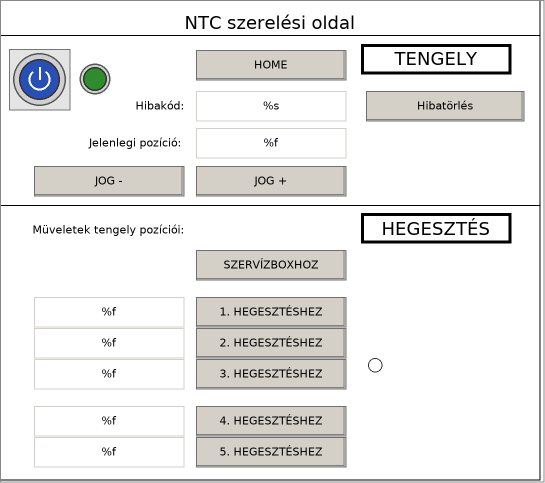
VISUALIZATION Hegesztes_Tengely_NTC  // 545x483
    Rectangle (0,0 540x480)
    PowerSwitch (9,49 61x61), variable: GVL.bJozsiServo, behaviour: TOGGLE, style: Switch-PowerSwitch-Blue
    Button (196,50 150x30), "HOME"
        OnMouseUp: execute { JOZSITENGELY.sJozsiAxisCommand:='HOME'; }
    Button (196,166 150x30), "JOG +"
        tap JOZSITENGELY.bJozsiJOGPlus
    Button (34,166 150x30), "JOG -"
        tap JOZSITENGELY.bJozsiJOGMinus
    Button (366,91 158x30), "Hibatörlés"
        tap JOZSITENGELY.bJozsiReset
    Textfield (196,91 150x30), "%s", text variable: JOZSITENGELY.nJozsiErrorCode, input disabled if: TRUE
    Label (34,128 150x30), "Jelenlegi pozíció:"
    Textfield (196,128 150x30), "%f", text variable: JOZSITENGELY.lrJozsiActPos, input disabled if: TRUE
    Textfield (34,297 150x30), "%f", text variable: GVL.lrHegesztoPosition1
        OnMouseClick: write the text variable via VisuDialogs.Numpad, min -10000, max -1
    Button (196,297 150x30), "1. HEGESZTÉSHEZ"
        OnMouseUp: execute { JOZSITENGELY.lrJozsiPosition:=GVL.lrHegesztoPosition1; JOZSITENGELY.sJozsiAxisCommand:='MOVE'; }
    RadioButton (366,249 177x232), variable: HEGESZTOK.nHegesztoNum
        Areas[0]: Text=Semelyik
        Areas[1]: Text=Program1HG1
        Areas[2]: Text=Program2HG1
        Areas[3]: Text=Program3HG1
        Areas[4]: Text=Program4HG2
        Areas[5]: Text=Program5HG2
        p340057476: Készenléti program
        p3123465237: 1. hegesztés program
        p2481256679: 2. hegesztés program
        p1032612214: 3. hegesztés program
        p3228930307: 4. hegesztés program
        p1847394450: 5. hegesztés program
        p1205187680: Program7HG3
        p3921487345: Program8HG3
    Textfield (34,328 150x30), "%f", text variable: GVL.lrHegesztoPosition2
        OnMouseClick: write the text variable via VisuDialogs.Numpad, min -10000, max -1
    Button (196,328 150x30), "2. HEGESZTÉSHEZ"
        OnMouseUp: execute { JOZSITENGELY.lrJozsiPosition:=GVL.lrHegesztoPosition2; JOZSITENGELY.sJozsiAxisCommand:='MOVE'; }
    Textfield (34,359 150x30), "%f", text variable: GVL.lrHegesztoPosition3
        OnMouseClick: write the text variable via VisuDialogs.Numpad, min -10000, max -1
    Button (196,359 150x30), "3. HEGESZTÉSHEZ"
        OnMouseUp: execute { JOZSITENGELY.lrJozsiPosition:=GVL.lrHegesztoPosition3; JOZSITENGELY.sJozsiAxisCommand:='MOVE'; }
    Textfield (34,406 150x30), "%f", text variable: GVL.lrHegesztoPosition4
        OnMouseClick: write the text variable via VisuDialogs.Numpad, min -10000, max -1
    Button (196,406 150x30), "4. HEGESZTÉSHEZ"
        OnMouseUp: execute { JOZSITENGELY.lrJozsiPosition:=GVL.lrHegesztoPosition4; JOZSITENGELY.sJozsiAxisCommand:='MOVE'; }
    Textfield (34,437 150x30), "%f", text variable: GVL.lrHegesztoPosition5
        OnMouseClick: write the text variable via VisuDialogs.Numpad, min -10000, max -1
    Button (196,437 150x30), "5. HEGESZTÉSHEZ"
        OnMouseUp: execute { JOZSITENGELY.lrJozsiPosition:=GVL.lrHegesztoPosition5; JOZSITENGELY.sJozsiAxisCommand:='MOVE'; }
    Button (196,250 150x30), "SZERVÍZBOXHOZ"
        OnMouseUp: execute { JOZSITENGELY.lrJozsiPosition:=GVL.lrNTCSzervizbox; JOZSITENGELY.sJozsiAxisCommand:='MOVE'; }
    Lamp1 (77,61 36x36), variable: JOZSITENGELY.bHomeReady, style: Lamp-Lamp1-Green
    Line (0,35) (540,35), "NTC szerelési oldal"
    Label (127,91 60x30), "Hibakód:"
    Line (0,205) (540,205)
    RoundedRectangle (361,44 150x30)
    Label (361,44 150x30), "TENGELY"
    RoundedRectangle (361,213 150x30)
    Label (361,214 150x30), "HEGESZTÉS"
    Label (27,215 163x30), "Müveletek tengely pozíciói:"
END_VISUALIZATION

(* stored: Version 1.1.0.1, ProductVersion 3.1.4024.11
   Visu Hegesztes_Tengely_NTC: Id {656f3d9a-1445-4901-a858-427525e75661} *)
